(* PLC project  *)

CONFIGURATION FSOE_IN
END_CONFIGURATION
